{attribute 'linkalways'} 
{attribute 'no_explicit_call' := 'This FB is a CLASS and must be accessed using methods or properties'}
{attribute 'enable_dynamic_creation'}
FUNCTION_BLOCK NodePrototypeHost IMPLEMENTS I_NodePrototypes
VAR
	prototypes : Dictionary;
	selfCreatedPrototypes : Stack;
END_VAR

METHOD PUBLIC Accept
VAR_INPUT
	visitor : I_NodePrototypeVisitor;
END_VAR
VAR
	enumerator : I_ForwardEnumerator;
	nodePrototype : I_NodePrototype;
END_VAR
enumerator := prototypes.GetEnumerator();

WHILE enumerator.MoveNext() DO
	
	IF enumerator.TryGet(nodePrototype) THEN
		nodePrototype.Accept(Visitor);
	END_IF

END_WHILE

enumerator.Dispose();
END_METHOD

METHOD AddNodeAsPrototype : I_NodePrototype
VAR_INPUT
	Path : T_MAXSTRING;
	Node : I_Node;
END_VAR
VAR
	prototype : I_NodePrototype;
END_VAR
prototype := CreatePrototype(Path, Node);
selfCreatedPrototypes.Push(prototype);
AddNodePrototype(prototype);
AddNodeAsPrototype := prototype;
END_METHOD

METHOD PUBLIC AddNodePrototype
VAR_INPUT
	NodePrototype : I_NodePrototype;
END_VAR
prototypes.AddOrUpdate(NodePrototype.Path, NodePrototype);
END_METHOD

METHOD PRIVATE CreatePrototype : I_NodePrototype
VAR_INPUT
	PrototypePath : T_MAXSTRING;
	PrototypeNode : I_Node;
END_VAR
VAR
	pNodePrototype : POINTER TO NodePrototype;
END_VAR
pNodePrototype := __NEW(NodePrototype(Path := PrototypePath, Node := PrototypeNode));
CreatePrototype := pNodePrototype^;
END_METHOD

METHOD PRIVATE DisposeSelfCreatedNodePrototypes : BOOL
VAR
	prototype : I_NodePrototype;
END_VAR
WHILE selfCreatedPrototypes.TryPop(prototype) DO
	prototype.Dispose();
END_WHILE
END_METHOD

METHOD FB_exit : BOOL
VAR_INPUT
	bInCopyCode : BOOL; // if TRUE, the exit method is called for exiting an instance that is copied afterwards (online change).
END_VAR
IF bInCopyCode THEN
	RETURN;
END_IF

DisposeSelfCreatedNodePrototypes();
END_METHOD

METHOD PUBLIC TryGetNodePrototypeByPath : BOOL
VAR_INPUT
	Path : T_MAXSTRING;
	Destination : REFERENCE TO I_NodePrototype;
END_VAR
VAR
	nodePrototype : I_NodePrototype;
END_VAR
IF NOT prototypes.TryGetValue(Path, nodePrototype) THEN
	RETURN;
END_IF

Destination := nodePrototype;
TryGetNodePrototypeByPath := TRUE;
END_METHOD

END_FUNCTION_BLOCK

(* stored: Version 1.1.0.1, ProductVersion 3.1.4024.12
   POU NodePrototypeHost: Id {0f3611b8-dc13-4989-9cc7-2b1a9dfa6a1b}, SpecialFunc None
   Folder Destructor: Id {11dfafd7-bfe1-4ac3-b221-2441d3673444}
   Folder Private: Id {f55cef08-2c4e-47c7-9688-2ca2e8391e35}
   Method Accept: Id {619b7ec2-3516-4862-b7fa-24a77dbc583a}
   Method AddNodeAsPrototype: Id {d6c829d7-eddc-47ad-bb68-526a309f1a6f}
   Method AddNodePrototype: Id {4d3a5f0c-8074-09fb-2906-a4aa05ab5434}
   Method CreatePrototype: Id {70bb490a-583f-43d4-9a69-6aeef34a308f}
   Method DisposeSelfCreatedNodePrototypes: Id {5ecc01e1-ef32-49f4-a9de-419a17111555}
   Method FB_exit: Id {7b52281d-300e-4a1e-be0b-45b74272fbb0}
   Method TryGetNodePrototypeByPath: Id {1552adb8-7411-41b6-a91a-3b378262f86b} *)
